{attribute 'qualified_only'}
{attribute 'strict'}
TYPE cResolvedDBStatusRoute :
(
	
	None := 0,
	Empty_NoRoute := 1,
	Empty_RoutedThisStation := 2,
	Empty_RoutedOtherStation := 3,
	Normal_RoutedThisStation := 5,
	Normal_RoutedOtherStation := 6,
	Normal_RoutedException := 7,
	Normal_RoutedConsolidation := 8,
	NonNormal_RoutedException := 9,
	UnknownDevice := 10,
	FastReceivingVision := 11,
	InvalidCombination := 12
	
) DINT;
END_TYPE

(* stored: Version 1.1.0.1, ProductVersion 3.1.4024.6
   DUT cResolvedDBStatusRoute: Id {741fe6bd-3f0b-44f4-9cbd-8ea6f1383484} *)
